// TIA Portal V18 program export: 1 tag tables, 0 data types, 0 data blocks, 2 code blocks (in call order from the OBs), 0 instance data blocks

VAR_GLOBAL   // PLC tag table "Default tag table"
   Tag_2 AT %MD50 : Real;
   Tag_3 AT %M40.0 : Bool;
END_VAR

ORGANIZATION_BLOCK "Main"   // OB1, LAD, ProgramCycle
TITLE = "Main Program Sweep (Cycle)"
{ S7_Optimized_Access := 'TRUE' }
VERSION : 0.1
// stored: AutoNumber true, IsIECCheckEnabled false, SetENOAutomatically false
   VAR_INPUT
      Initial_Call : Bool;   // Initial call of this OB
      Remanence : Bool;   // =True, if remanent data are available
   END_VAR
   VAR_TEMP
      temp_R : Real;
      temp_Rg : Real;
      temp_W : Word;
      temp_Rg1 : Real;
      temp_Rg2_1 : Real;
      temp_Rg3_1 : Real;
      temp_Rg3_2 : Real;
      temp_real : Real;
      temp_real_1 : Real;
      temp_real_2 : Real;
      temp_real_3 : Real;
      temp_real_4 : Real;
      temp_real_5 : Real;
      temp_real_6 : Real;
      temp_real_7 : Real;
      temp_real_8 : Real;
      temp_real_9 : Real;
      temp_B : Bool;
      temp_start : Bool;
      temp_Rg2 : Real;
      temp_W1 : Int;
      temp_Rg3 : Real;
      Param_SetBit_0 : Bool;
      Param_SetBit_1 : Bool;
   END_VAR
BEGIN

REGION Network 2
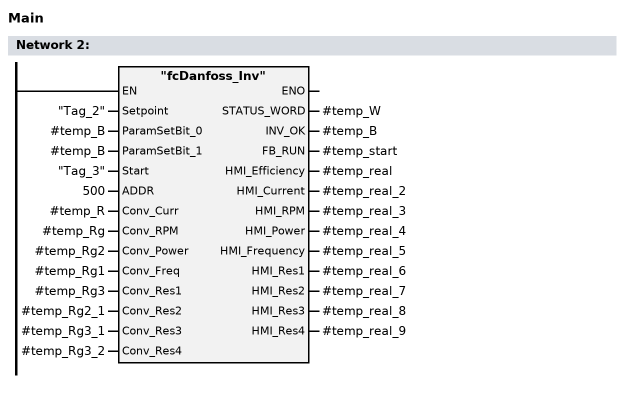
   RUNG wire#powerrail
      "fcDanfoss_Inv"(Setpoint := "Tag_2", ParamSetBit_0 := #temp_B, ParamSetBit_1 := #temp_B, Start := "Tag_3", ADDR := 500, Conv_Curr := #temp_R, Conv_RPM := #temp_Rg, Conv_Power := #temp_Rg2, Conv_Freq := #temp_Rg1, Conv_Res1 := #temp_Rg3, Conv_Res2 := #temp_Rg2_1, Conv_Res3 := #temp_Rg3_1, Conv_Res4 := #temp_Rg3_2, STATUS_WORD => #temp_W, INV_OK => #temp_B, FB_RUN => #temp_start, HMI_Efficiency => #temp_real, HMI_Current => #temp_real_2, HMI_RPM => #temp_real_3, HMI_Power => #temp_real_4, HMI_Frequency => #temp_real_5, HMI_Res1 => #temp_real_6, HMI_Res2 => #temp_real_7, HMI_Res3 => #temp_real_8, HMI_Res4 => #temp_real_9)
   END_RUNG
   // the same network as SCL:
   "fcDanfoss_Inv"(Setpoint := "Tag_2",
                   ParamSetBit_0 := #temp_B,
                   ParamSetBit_1 := #temp_B,
                   Start := "Tag_3",
                   ADDR := 500,
                   Conv_Curr := #temp_R,
                   Conv_RPM := #temp_Rg,
                   Conv_Power := #temp_Rg2,
                   Conv_Freq := #temp_Rg1,
                   Conv_Res1 := #temp_Rg3,
                   Conv_Res2 := #temp_Rg2_1,
                   Conv_Res3 := #temp_Rg3_1,
                   Conv_Res4 := #temp_Rg3_2,
                   STATUS_WORD => #temp_W,
                   INV_OK => #temp_B,
                   FB_RUN => #temp_start,
                   HMI_Efficiency => #temp_real,
                   HMI_Current => #temp_real_2,
                   HMI_RPM => #temp_real_3,
                   HMI_Power => #temp_real_4,
                   HMI_Frequency => #temp_real_5,
                   HMI_Res1 => #temp_real_6,
                   HMI_Res2 => #temp_real_7,
                   HMI_Res3 => #temp_real_8,
                   HMI_Res4 => #temp_real_9);
END_REGION

REGION Network 3
   // Test network
END_REGION
END_ORGANIZATION_BLOCK

FUNCTION "Test" : Void   // FC1, STL
{ S7_Optimized_Access := 'TRUE' }
VERSION : 0.1
// stored: AutoNumber true, UDAEnableTagReadback false
BEGIN

NETWORK
TITLE = 
      NOP   0;

END_FUNCTION
